TYPE "Prg_Pivot"
VERSION : 0.1
// Block: Prg_Pivot
   STRUCT
      PrgNo : DInt;
      PrgName : "String[30]";
      RecordNo : Int;
   END_STRUCT;

END_TYPE
